(*			
	RAFALOS
	Rafał Osajda		19.09.2025		TC 4024.66
	FB Bazowy dla wszystkich elementów złożonych
*)
FUNCTION_BLOCK FB_BaseGroupElement EXTENDS FB_BaseControlElement IMPLEMENTS ITF_BaseGroupElement, ITF_BaseGroupElement_HMI_Connector,
 		ITF_BaseMessengerRecipient, ITF_BaseMessengerSender
VAR
	arrControlElement			: ARRAY [1..GVL_BaseConstans.MAX_ITEM_PER_ELEMENT] OF ITF_BaseControlElement;
	uiNumberOfControlElement	: UINT;
	itfCommunicator				: ITF_BaseCommunicator;
END_VAR

METHOD PROTECTED AddControlElement : BOOL
VAR_INPUT
	itfControlElement		: ITF_BaseControlElement;
END_VAR
IF (THIS^.uiNumberOfControlElement + 1 <= GVL_BaseConstans.MAX_ITEM_PER_ELEMENT) THEN
	THIS^.uiNumberOfControlElement		:= THIS^.uiNumberOfControlElement + 1;
	THIS^.arrControlElement [THIS^.uiNumberOfControlElement]	:= itfControlElement;
	AddControlElement			:= TRUE;
ELSE
	;//zwrocenie zbyt dużo komponentow
END_IF
END_METHOD

METHOD PUBLIC ConfirmReceipt : BOOL
VAR_INPUT
	sText: STRING;
END_VAR
ConfirmReceipt	:= THIS^.itfCommunicator.ReceiveDataConfirm (sText := sText, itfRecipient := THIS^);
END_METHOD

(*			
	RafalOS
	Rafał Osajda		27.03.2025		TC 4024.66
	Obsluga bledow sprawdzanie czy jakis blad sie nei pojawil i ustawienie stanu lub wylaczenie
*)
METHOD PUBLIC ExecuteEveryCycle_Error
VAR
	iI					: INT;
END_VAR
SUPER^.ExecuteEveryCycle_Error ();

FOR iI := 1 TO TO_INT (THIS^.uiNumberOfControlElement) DO
	THIS^.arrControlElement [iI].ExecuteEveryCycle_Error ();
END_FOR
END_METHOD

(*			
	RafalOS
	Rafał Osajda		27.03.2025		TC 4024.66
	Wywolanie co cykl operacji 
*)
METHOD PUBLIC ExecuteEveryCycle_Operation
VAR
	iI				: INT;
END_VAR
SUPER^.ExecuteEveryCycle_Operation ();

FOR iI := 1 TO TO_INT (THIS^.uiNumberOfControlElement) DO
	THIS^.arrControlElement [iI].ExecuteEveryCycle_Operation ();
END_FOR
END_METHOD

(*			
	RafalOS
	Rafał Osajda		27.03.2025		TC 4024.66
	Aktualizacja flag 
*)
METHOD PUBLIC ExecuteEveryCycle_Status
VAR
	iI				: INT;
END_VAR
SUPER^.ExecuteEveryCycle_Status ();

FOR iI := 1 TO TO_INT (THIS^.uiNumberOfControlElement) DO
	THIS^.arrControlElement [iI].ExecuteEveryCycle_Status ();
END_FOR
END_METHOD

(*			
	RafalOS
	Rafał Osajda		27.03.2025		TC 4024.66
	Testowanie czy nei pojawil sie jakis rozkaz i uruchomienie odpowiednich operacji
*)
METHOD PUBLIC ExecuteEveryCycle_Test
VAR
	iI			: INT;
END_VAR
SUPER^.ExecuteEveryCycle_Test ();

FOR iI := 1 TO TO_INT (THIS^.uiNumberOfControlElement) DO
	THIS^.arrControlElement [iI].ExecuteEveryCycle_Test ();
END_FOR
END_METHOD

METHOD FB_init : BOOL
VAR_INPUT
	bInitRetains : BOOL; // if TRUE, the retain variables are initialized (warm start / cold start)
	bInCopyCode : BOOL;  // if TRUE, the instance afterwards gets moved into the copy code (online change)
END_VAR
THIS^.stIdentifier.eType			:= E_BaseElementType.eGroup;
END_METHOD

METHOD PUBLIC FirstCycle : BOOL
VAR_INPUT
END_VAR
VAR
	bResult			: bool;
	iI				: INT;
END_VAR
bResult				:= SUPER^.FirstCycle ();

FOR iI := 1 TO TO_INT (THIS^.uiNumberOfControlElement) DO
	bResult			:= bResult AND THIS^.arrControlElement [iI].FirstCycle ();
END_FOR

FirstCycle			:= bResult;
END_METHOD

METHOD GetITFGroupElement : ITF_BaseGroupElement
VAR_INPUT
END_VAR
GetITFGroupElement	:= THIS^;
END_METHOD

METHOD GetITFTopElement : ITF_BaseTopElement
VAR_INPUT
END_VAR
GetITFTopElement		:= null;
END_METHOD

(*			
	RafalOS
	Rafał Osajda		27.05.2025		TC 4024.66
	Metoda bazowania kontrektnego elementu 
*)
METHOD PROTECTED HomingCycle : BOOL
VAR
	iI			: INT;
END_VAR
CASE THIS^.stHoming.iElementHomingStep OF
0	:
	FOR iI := 1 TO TO_INT (THIS^.uiNumberOfControlElement) DO
		THIS^.arrControlElement [iI].HomingStart ();
	END_FOR
	THIS^.stHoming.iElementHomingStep	:= THIS^.stHoming.iElementHomingStep + 10;
	HomingCycle							:= TRUE;
10	:
	THIS^.stHoming.iElementHomingStep	:= THIS^.stHoming.iElementHomingStep + 10;
	HomingCycle							:= TRUE;
20	:
	IF (THIS^.HomingGetDone ()) THEN
		THIS^.stHoming.iElementHomingStep 	:= GVL_BaseConstans.FINISH_STEP;
	END_IF	
	HomingCycle							:= TRUE;
GVL_BaseConstans.FINISH_STEP :
	HomingCycle							:= FALSE;
END_CASE
END_METHOD

(*			
	RafalOS
	Rafał Osajda		31.03.2025		TC 4024.66
	Flaga że w tej sesji pracy maszyny element został już wybazowany
*)
METHOD PUBLIC HomingGetDone : BOOL
VAR
	iI				: INT;
	btmpHomingDone	: BOOL;
END_VAR
btmpHomingDone		:= TRUE;
FOR iI := 1 TO TO_INT (THIS^.uiNumberOfControlElement) DO
	btmpHomingDone	:= btmpHomingDone AND THIS^.arrControlElement [iI].HomingGetDone ();
	IF (NOT btmpHomingDone) THEN
		EXIT;
	END_IF
END_FOR
HomingGetDone		:= btmpHomingDone;
END_METHOD

(*			
	RafalOS
	Rafał Osajda		11.04.2025		TC 4024.66
	Zwraca czy bazowanie jest potrzebne
*)
METHOD PUBLIC HomingGetIsNeeded : BOOL
VAR
	btmpHomingIsNeeded	: BOOL := FALSE;
	iI					: INT;
END_VAR
FOR iI := 1 TO TO_INT (THIS^.uiNumberOfControlElement) DO
	btmpHomingIsNeeded	:= btmpHomingIsNeeded OR THIS^.arrControlElement [iI].HomingGetIsNeeded ();
	IF (btmpHomingIsNeeded) THEN
		EXIT;
	END_IF
END_FOR
HomingGetIsNeeded		:= btmpHomingIsNeeded;
END_METHOD

(*			
	RafalOS
	Rafał Osajda		30.04.2025		TC 4024.66
	Zwraca czy element jest czymś zajety
*)
METHOD PUBLIC IsDoNothing : BOOL
VAR
	iI				: INT;
	btmpDoNothing	: BOOL := TRUE;
END_VAR
FOR iI := 1 TO TO_INT (THIS^.uiNumberOfControlElement) DO
	btmpDoNothing		:= btmpDoNothing AND THIS^.arrControlElement [iI].IsDoNothing ();
	IF (NOT btmpDoNothing) THEN
		EXIT;
	END_IF
END_FOR
THIS^.bDoNothing		:= btmpDoNothing;
IsDoNothing			:= btmpDoNothing;
END_METHOD

(*			
	RafalOS
	Rafał Osajda		30.04.2025		TC 4024.66
	Zwraca czy element jest w pozycji 0 - referencyjnej
*)
METHOD PUBLIC IsPosition0 : BOOL
VAR
	iI					: INT;
	btmpPosition0		: BOOL;
END_VAR
FOR iI := 1 TO TO_INT (THIS^.uiNumberOfControlElement) DO
	btmpPosition0		:= btmpPosition0 AND THIS^.arrControlElement [iI].IsPosition0 ();
	IF (NOT btmpPosition0) THEN
		EXIT;
	END_IF
END_FOR
THIS^.bPosition0		:= btmpPosition0;
IsPosition0			:= btmpPosition0;
END_METHOD

METHOD PUBLIC IsValidCommonData : BOOL
VAR_INPUT
END_VAR

VAR
	bResult: BOOL;
	iI: INT;
END_VAR
bResult						:= SUPER^.IsValidCommonData ();

FOR iI := 1 TO TO_INT (THIS^.uiNumberOfControlElement) DO
	bResult					:= bResult AND THIS^.arrControlElement [iI].IsValidCommonData ();
END_FOR

IsValidCommonData			:= bResult;
END_METHOD

(*			
	RafalOS
	Rafał Osajda		07.10.2025		TC 4024.66
	Dodpisywanie się do listy logera
*)
METHOD PUBLIC JoinTheLogger : BOOL
VAR_INPUT
END_VAR

VAR
	bResult: BOOL;
	iI: INT;
END_VAR
bResult			:= SUPER^.JoinTheLogger ();

FOR iI := 1 TO  TO_INT (THIS^.uiNumberOfControlElement) DO
	bResult 	:= bResult AND THIS^.arrControlElement [iI].JoinTheLogger ();
END_FOR

JoinTheLogger	:= bResult;
END_METHOD

METHOD PUBLIC LinkCommonData : BOOL
VAR_INPUT
	stCommonData				: REFERENCE TO ST_BaseCommonData;
END_VAR
VAR
	bResult						: BOOL;
	iI: INT;
END_VAR
bResult							:= SUPER^.LinkCommonData (stCommonData := stCommonData);

FOR iI := 1 TO TO_INT (THIS^.uiNumberOfControlElement) DO
	bResult := bResult AND THIS^.arrControlElement [iI].LinkCommonData (stCommonData := stCommonData);
END_FOR

LinkCommonData					:= bResult;
END_METHOD

METHOD PUBLIC LinkCommunicator : BOOL
VAR_INPUT
	fbCommunicator				: ITF_BaseCommunicator;
END_VAR
THIS^.itfCommunicator			:= fbCommunicator;
IF (THIS^.itfCommunicator <> 0) THEN
	LinkCommunicator			:= TRUE;
END_IF
END_METHOD

METHOD PUBLIC LinkSS1 : BOOL
VAR_INPUT
	fbSS1			: ITF_BaseFlagGet;
END_VAR

VAR
	bresult: BOOL;
	iI: INT;
END_VAR
bresult				:= SUPER^.LinkSS1 (fbSS1 := fbSS1);

FOR iI := 1 TO TO_INT (THIS^.uiNumberOfControlElement) DO
	bresult			:= bresult AND THIS^.arrControlElement [iI].LinkSS1 (fbSS1	:= fbSS1);
END_FOR

LinkSS1				:= bresult;
END_METHOD

METHOD PUBLIC LinkSTO : BOOL
VAR_INPUT
	fbSTO			: ITF_BaseFlagGet;
END_VAR

VAR
	bresult: BOOL;
	iI: INT;
END_VAR
bresult				:= SUPER^.LinkSTO (fbSTO := fbSTO);

FOR iI := 1 TO TO_INT (THIS^.uiNumberOfControlElement) DO
	bresult			:= bresult AND THIS^.arrControlElement [iI].LinkSTO (fbSTO	:= fbSTO);
END_FOR

LinkSTO				:= bresult;
END_METHOD

METHOD PROTECTED PowerOffCycle : BOOL
VAR
	iI							: INT;
	bPowerStatus			: BOOL;
END_VAR
CASE stPower.cmdTurnOff.GetStep () OF
0	:
	FOR iI := 1 TO TO_INT (THIS^.uiNumberOfControlElement) DO
		THIS^.arrControlElement [iI].PowerTurnOff ();
	END_FOR
	THIS^.stPower.cmdTurnOff.SetStepINC10 ();
	PowerOffCycle			:= TRUE;
10	:
	bPowerStatus			:= FALSE;
	FOR iI := 1 TO TO_INT (THIS^.uiNumberOfControlElement) DO
		bPowerStatus		:= bPowerStatus OR THIS^.arrControlElement [iI].PowerGetStatus ();
		IF (bPowerStatus) THEN
			EXIT;
		END_IF
	END_FOR	
	IF (NOT bPowerStatus) THEN
		THIS^.stPower.bStatus	:= FALSE;
		THIS^.stPower.cmdTurnOff.SetStepAsFinal ();
	ELSE
		PowerOffCycle			:= TRUE;
	END_IF	
END_CASE
END_METHOD

METHOD PROTECTED PowerOnCycle : BOOL
VAR
	iI						: INT;
	bPowerStatus		: BOOL;
END_VAR
CASE stPower.cmdTurnOn.GetStep () OF
0	:
	FOR iI := 1 TO TO_INT (THIS^.uiNumberOfControlElement) DO
		THIS^.arrControlElement [iI].PowerTurnOn ();
	END_FOR
	THIS^.stPower.cmdTurnOn.SetStepINC10 ();
	PowerOnCycle				:= TRUE;
10	:
	bPowerStatus			:= TRUE;
	FOR iI := 1 TO TO_INT (THIS^.uiNumberOfControlElement) DO
		bPowerStatus		:= bPowerStatus AND THIS^.arrControlElement [iI].PowerGetStatus ();
		IF (NOT bPowerStatus) THEN
			EXIT;
		END_IF
	END_FOR	
	IF (bPowerStatus) THEN
		THIS^.stPower.bStatus	:= TRUE;
		THIS^.stPower.cmdTurnOn.SetStepAsFinal ();
		PowerOnCycle			:= FALSE;
	ELSE
		PowerOnCycle			:= TRUE;
	END_IF	
END_CASE
END_METHOD

METHOD PUBLIC Receive_BOOL : BOOL
VAR_INPUT
	sText		: STRING;
END_VAR
VAR_OUTPUT
	bValue		: BOOL;	
END_VAR
Receive_BOOL			:= THIS^.itfCommunicator.ReceiveData_BOOL (sText := sText, itfRecipient := THIS^, bValue => bValue);
END_METHOD

METHOD PUBLIC Receive_REAL : BOOL
VAR_INPUT
	sText		: STRING;
END_VAR
VAR_OUTPUT
	rValue		: REAL;	
END_VAR
Receive_REAL			:=  THIS^.itfCommunicator.ReceiveData_REAL (sText := sText, itfRecipient := THIS^, rValue => rValue);
END_METHOD

METHOD PROTECTED ResetOperation : BOOL
VAR
	bResult				: BOOL;
END_VAR
bResult					:= SUPER^.ResetOperation ();


ResetOperation			:= FALSE OR bResult;
END_METHOD

METHOD Send_BOOL : BOOL
VAR_INPUT
	sText				: STRING;
END_VAR
Send_BOOL		:= THIS^.itfCommunicator.SendData_BOOL (sText := sText, itfSender := THIS^);
END_METHOD

METHOD Send_REAL : BOOL
VAR_INPUT
	sText		: STRING;
	rValue		: REAL;
END_VAR
Send_REAL			:= THIS^.itfCommunicator.SendData_REAL (sText := sText, rValue := rValue, itfSender := THIS^);
END_METHOD

METHOD PUBLIC SetCode
VAR_INPUT
	sCode							: STRING;
	sAdd							: STRING;
END_VAR
VAR
	sItemCode						: STRING;
	iI								: INT;
	sParentCode						: STRING;
	arrSegment						: ARRAY [0..GVL_BaseConstans.MAX_NESTING_LEVEL] OF STRING;
	iDotPosition					: INT;
	iLast							: INT;
	
END_VAR
//sKodRodzica	:=  UtworzKodElementu (sKodRodzica := sKod, sDopisz := TO_STRING (THIS^.zwrocID ()));
SUPER^.SetCode (sCode := sCode, sAdd := sAdd);
sParentCode						:= THIS^.GetCode ();

IF (THIS^.uiNumberOfComponents > 0) THEN
	arrSegment [0]				:= THIS^.arrComponent [THIS^.uiNumberOfComponents].GetCode ();
	FOR iI := 1 TO TO_INT (GVL_BaseConstans.MAX_NESTING_LEVEL) DO
		iDotPosition			:= find (STR1 := arrSegment [0], STR2 := '.');
		IF (iDotPosition = 0) THEN
			arrSegment [iI]	:= arrSegment [0];
			EXIT;
		ELSE
			arrSegment [iI]		:= Tc2_Standard.LEFT (STR := arrSegment [0], SIZE := iDotPosition - 1);
			arrSegment [0]		:= Tc2_Standard.DELETE (STR := arrSegment [0], POS := 1, LEN := iDotPosition);
		END_IF
	END_FOR
	FOR iI := 0 TO TO_INT (GVL_BaseConstans.MAX_NESTING_LEVEL) - 1 DO
		IF (TO_INT (arrSegment [TO_INT (GVL_BaseConstans.MAX_NESTING_LEVEL) - iI]) <> 0 ) THEN
			iLast			:= TO_INT (arrSegment [TO_INT (GVL_BaseConstans.MAX_NESTING_LEVEL) - iI]);
			EXIT;
		END_IF
	END_FOR
END_IF

FOR iI := 1 TO TO_INT (THIS^.uiNumberOfControlElement) DO
//	sKodKomponentu	:= UtworzKodElementu (sKodRodzica := sKod, sDopisz := TO_STRING (iI));
	THIS^.arrControlElement [iI].SetCode (sCode	:= sParentCode, sAdd := TO_STRING (iI + iLast));
END_FOR
END_METHOD

(*			
	RafalOS
	Rafał Osajda		03.10.2025		TC 4024.66
	nadawanie unikalnych ID dla zdarzeń
*)
METHOD PUBLIC SetEventsIDs : UINT
VAR_INPUT
	uiNewID		: UINT;
END_VAR
VAR
	iI			: INT;
	uiLastID	: UINT;
END_VAR
uiLastID		:= SUPER^.SetEventsIDs (uiNewID	:= uiNewID);

FOR iI := 1 TO TO_INT (THIS^.uiNumberOfControlElement) DO 
	uiLastID			:= THIS^.arrControlElement [iI].SetEventsIDs (uiNewID	:= uiLastID);
END_FOR
SetEventsIDs				:= uiLastID;
END_METHOD

METHOD PUBLIC SetID : UINT
VAR_INPUT
	uiID					: UINT;
END_VAR
VAR
	uiLastID				: UINT;
	iI						: INT;
END_VAR
uiLastID				:= SUPER^.SetID (uiID	:= uiID);

FOR iI := 1 TO TO_INT (THIS^.uiNumberOfControlElement) DO 
	uiLastID			:= THIS^.arrControlElement [iI].SetID (uiID	:= uiLastID + 1);
END_FOR
SetID					:= uiLastID;
END_METHOD

END_FUNCTION_BLOCK

(* stored: Version 1.1.0.1
   POU FB_BaseGroupElement: Id {1f8518b0-2e03-0c13-2a4a-ffc3b6f9b887}, SpecialFunc None
   Folder Bazowanie: Id {ac03e261-94f6-0d08-2b29-69a0f6f80414}
   Folder Events: Id {20f6f417-5dd7-052c-022d-8978faa14be3}
   Folder ID: Id {9d43db93-a825-0ef2-1289-7c7210b94e63}
   Folder ITF_BaseComponent: Id {21d91ff8-321c-0a3c-3e32-f71a83cd7a28}
   Folder ITF_BaseControlElement: Id {7a13d05e-a071-0aa3-2f07-a3977bd5f5b3}
   Folder ITF_DecoratedElement: Id {a1479acc-3f0a-0c64-3109-7e2e716b7d21}
   Folder Komunikator: Id {437b8f14-4a81-003f-095e-33d967fc7cb0}
   Folder Reset: Id {f175fff7-b28d-0fc9-2a54-b324df7e3bfb}
   Folder WiazanieZmiennych: Id {2b50b030-a9ec-06ce-1ddf-f0356b93fad0}
   Folder Zasilanie: Id {27dafdd4-57cf-0313-207b-208322f99c30}
   Method AddControlElement: Id {175b37ba-638b-0727-26cf-573800512486}
   Method ConfirmReceipt: Id {600100d4-0187-08ab-39be-f426b6343e54}
   Method ExecuteEveryCycle_Error: Id {27999fb5-d889-03ba-3e6e-c89cb8983a76}
   Method ExecuteEveryCycle_Operation: Id {9b6c22a1-ff3d-0cb3-36d0-b2883b8e1ec9}
   Method ExecuteEveryCycle_Status: Id {697110ad-2da0-0583-304b-85b1ad08e3bb}
   Method ExecuteEveryCycle_Test: Id {879f7bc3-0f18-0b43-0dc5-691b7892df40}
   Method FB_init: Id {a18f7400-8689-05ae-3b31-59cab5e8ddb8}
   Method FirstCycle: Id {fede4491-2815-0c5d-25f3-a52cafaf5311}
   Method GetITFGroupElement: Id {d5980707-73de-0a3f-2ced-ebfc86d9bd9f}
   Method GetITFTopElement: Id {d653e274-f203-086f-3196-94fdc98a5300}
   Method HomingCycle: Id {5fc8b8d1-8229-0a71-1575-f7bc7c0780a2}
   Method HomingGetDone: Id {f022fc44-c924-0052-0029-05a35ee9823e}
   Method HomingGetIsNeeded: Id {1f91511b-58bd-09d6-1a5a-e46fda26b3f4}
   Method IsDoNothing: Id {f182bed7-6e94-09dd-3b80-e6560a2640bc}
   Method IsPosition0: Id {71e3e5d7-b708-0c78-3ca1-830cdfe03509}
   Method IsValidCommonData: Id {f68feac5-aff9-07a7-017f-3067903007ab}
   Method JoinTheLogger: Id {63b62d03-fe40-084c-0b22-a3d0bbf0b2bf}
   Method LinkCommonData: Id {163c9121-a3cf-0bfe-2517-ea6f42e3be4a}
   Method LinkCommunicator: Id {9a87eb73-fc46-0627-0754-c3115bdb72cb}
   Method LinkSS1: Id {76e517ec-0eff-075d-0625-cf0f5460cacb}
   Method LinkSTO: Id {91e2e203-b610-04e4-1b52-ed4f584923fa}
   Method PowerOffCycle: Id {418e83ec-8f97-07d4-0867-9ef529a73ef8}
   Method PowerOnCycle: Id {08b33ced-f9ae-0bb9-1205-79dbe801e4dd}
   Method Receive_BOOL: Id {c8be6563-f9ac-0fe3-080e-4719d4e50552}
   Method Receive_REAL: Id {ca20180b-24f1-056a-188c-82d969f44ae2}
   Method ResetOperation: Id {b6491d3e-1705-00b0-1aa1-54f9fbb764a3}
   Method Send_BOOL: Id {117b18b6-429b-04be-05c3-fe2b74a629c9}
   Method Send_REAL: Id {3eaba51e-2f11-0c9c-3a2f-6ac261cce02a}
   Method SetCode: Id {3432e546-4149-00a7-0fb9-e73b7e1c9dbd}
   Method SetEventsIDs: Id {0185e120-5cb8-0dba-3756-ff856ef7df3c}
   Method SetID: Id {fea103d8-a0ad-03db-1bf2-3008a70fc842} *)
